FUNCTION_BLOCK fb_gm_operationEjector
VAR_INPUT
END_VAR
VAR_OUTPUT
END_VAR
VAR
	SFCInit : bool;
	flgInitDone: BOOL;
	trn_vacuumOnDone: BOOL;
	trn_vacuumOffDone: BOOL;
	trn_breakOnDone: BOOL;
	trn_breakOffDone: BOOL;
	var_process: INT;
END_VAR

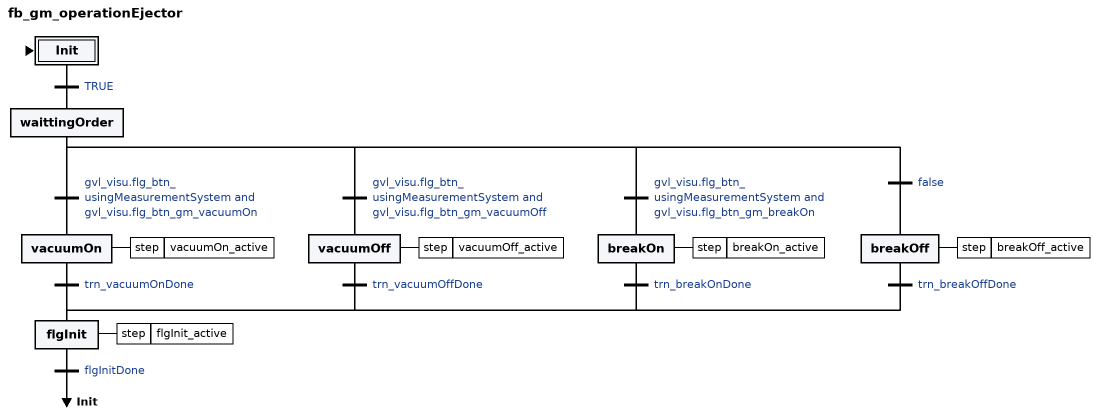
INITIAL_STEP Init:
END_STEP
TRANSITION FROM Init TO waittingOrder
    := TRUE;
END_TRANSITION
STEP waittingOrder:
END_STEP
TRANSITION FROM waittingOrder TO vacuumOn
    := gvl_visu.flg_btn_usingMeasurementSystem and gvl_visu.flg_btn_gm_vacuumOn;
END_TRANSITION
STEP vacuumOn:
    vacuumOn_active(N);  // step action
END_STEP
TRANSITION FROM vacuumOn TO flgInit
    := trn_vacuumOnDone;
END_TRANSITION
TRANSITION FROM waittingOrder TO vacuumOff
    := gvl_visu.flg_btn_usingMeasurementSystem and gvl_visu.flg_btn_gm_vacuumOff;
END_TRANSITION
STEP vacuumOff:
    vacuumOff_active(N);  // step action
END_STEP
TRANSITION FROM vacuumOff TO flgInit
    := trn_vacuumOffDone;
END_TRANSITION
TRANSITION FROM waittingOrder TO breakOn
    := gvl_visu.flg_btn_usingMeasurementSystem and gvl_visu.flg_btn_gm_breakOn;
END_TRANSITION
STEP breakOn:
    breakOn_active(N);  // step action
END_STEP
TRANSITION FROM breakOn TO flgInit
    := trn_breakOnDone;
END_TRANSITION
TRANSITION FROM waittingOrder TO breakOff
    := false;
END_TRANSITION
STEP breakOff:
    breakOff_active(N);  // step action
END_STEP
TRANSITION FROM breakOff TO flgInit
    := trn_breakOffDone;
END_TRANSITION
STEP flgInit:
    flgInit_active(N);  // step action
END_STEP
TRANSITION FROM flgInit TO Init
    := flgInitDone;
END_TRANSITION

ACTION breakOff_active:
IF breakOff._x AND breakOff.x = FALSE THEN
	trn_breakOffDone := FALSE;
	gvl_solv.fbi_gm_ejector.in_flg_run := FALSE;
	gvl_solv.fbi_gm_ejector.in_var_vacMode := eP_ejevacMode.breakOff;
	var_process := 0;
ELSIF breakOff._x AND breakOff.x THEN
	CASE var_process OF
		0:
			gvl_solv.fbi_gm_ejector.in_flg_run := TRUE;
			var_process := 0;
		1:
			IF gvl_solv.fbi_gm_ejector.out_flg_Done THEN
				gvl_solv.fbi_gm_ejector.in_flg_run := FALSE;
				trn_breakOffDone := TRUE;
			END_IF
	END_CASE
END_IF
END_ACTION

ACTION breakOn_active:
IF breakOn._x AND breakOn.x = FALSE THEN
	trn_breakOnDone := FALSE;
	gvl_solv.fbi_gm_ejector.in_flg_run := FALSE;
	gvl_solv.fbi_gm_ejector.in_var_vacMode := eP_ejevacMode.break;
	var_process := 0;
ELSIF breakOn._x AND breakOn._x THEN
	CASE var_process OF
		0:
			gvl_solv.fbi_gm_ejector.in_flg_run := TRUE;
			var_process := 1;
		1:
			IF gvl_solv.fbi_gm_ejector.out_flg_Done THEN
				gvl_solv.fbi_gm_ejector.in_flg_run := FALSE;
				trn_breakOnDone := TRUE;
			END_IF
	END_CASE
END_IF
END_ACTION

ACTION flgInit_active:
IF flgInit._x AND flgInit.x = FALSE THEN
	flgInitDone := FALSE;
	gvl_visu.flg_btn_gm_vacuumOn := FALSE;
	gvl_visu.flg_btn_gm_vacuumOff := FALSE;
	gvl_visu.flg_btn_gm_breakOn := FALSE;
	
ELSIF flgInit._x AND flgInit.x THEN
	flgInitDone := TRUE;
END_IF
END_ACTION

PROPERTY p_Init : bool
GET
p_init := THIS^.SFCInit;
END_GET
SET
THIS^.SFCInit := p_Init;
END_SET
END_PROPERTY

ACTION vacuumOff_active:
IF vacuumOff._x AND vacuumOff.x = FALSE THEN
	trn_vacuumOffDone := FALSE;
	gvl_solv.fbi_gm_ejector.in_flg_run := FALSE;
	gvl_solv.fbi_gm_ejector.in_var_vacMode := eP_ejevacMode.vacOff;
	var_process := 0;
ELSIF vacuumOff._x AND vacuumOff.x THEN
	CASE var_process OF
		0:
			gvl_solv.fbi_gm_ejector.in_flg_run := TRUE;
			var_process := 1;
		1:
			IF gvl_solv.fbi_gm_ejector.out_flg_Done THEN
			gvl_solv.fbi_gm_ejector.in_flg_run := FALSE;
			trn_vacuumOffDone := TRUE;
		END_IF
	END_CASE
END_IF
END_ACTION

ACTION vacuumOn_active:
IF vacuumOn._x AND vacuumOn.x = FALSE THEN
	trn_vacuumOnDone := FALSE;
	gvl_solv.fbi_gm_ejector.in_flg_run := FALSE;
	gvl_solv.fbi_gm_ejector.in_var_vacMode := eP_ejevacMode.halt;
	var_process := 0;
ELSIF vacuumOn._x AND vacuumOn.x THEN
	CASE var_process OF
		0:
			gvl_solv.fbi_gm_ejector.in_flg_run := TRUE;
			var_process := 1;
		1:
			IF gvl_solv.fbi_gm_ejector.out_flg_Done THEN
				gvl_solv.fbi_gm_ejector.in_flg_run := FALSE;
				trn_vacuumOnDone := TRUE;
			END_IF
	END_CASE
END_IF
END_ACTION

END_FUNCTION_BLOCK

(* stored: Version 1.1.0.1, ProductVersion 3.1.4024.11
   POU fb_gm_operationEjector: Id {4fd524cc-6f26-4953-afa7-e12a0e828e5d}, SpecialFunc None
   Action breakOff_active: Id {e90dac4c-42ed-4e4e-8ac4-a0ac3c537040}
   Action breakOn_active: Id {04b8a6cb-2c93-46e1-97c5-91dde109138d}
   Action flgInit_active: Id {9d621d44-e77a-4120-bd09-0ea994644392}
   Property p_Init: Id {0255b3f9-3409-4c29-a6cf-f6ceb2387610}
   Get Get: Id {f9c6077a-efd4-4b2f-ab05-6a3b91a4f085}
   Set Set: Id {c693b359-2beb-4c1e-9048-e645a01e97e7}
   Action vacuumOff_active: Id {8fc7bd4e-b3e9-4ec4-806b-36f64a2b3240}
   Action vacuumOn_active: Id {7660cc48-ca28-4f6a-b0fc-63d055be4611} *)
